PROGRAM Encoder
VAR
	//Encoder1 : Link to EL5001
	nRawData 		: REAL;
	nScaling 		: REAL;
	nOffset 		: REAL;
	nVoltage 		: REAL;
	testEncoder		: sEncoder;
	sScalingTable 	: ARRAY[0..2] OF WSTRING := ["Stacker Table WAN", "WT3 WAN"];
	iScaleTable		: INT := 0;
END_VAR



IF iScaleTable=0 THEN
	nScaling := 0.0004224;
ELSIF  iScaleTable=1 THEN
	nScaling := 0.0002636080;
ELSE
	nScaling := 0.0004224;
END_IF
 
//nCounter := UDINT_TO_REAL(Encoder1.
//testEncoder.bInputToggle := TRUE;
nVoltage := UDINT_TO_REAL(testEncoder.uCounter) * nScaling + nOffset;
	
(*
IF Module_IO.iBypassSwitch THEN
	testEncoder.bInputToggle := TRUE;
	nVoltage := UDINT_TO_REAL(testEncoder.uCounter) * nScaling;
ELSE
	testEncoder.bInputToggle := FALSE;
END_IF
*)

END_PROGRAM

(* stored: Version 1.1.0.1, ProductVersion 3.1.4024.11
   POU Encoder: Id {30275c88-29ac-483c-a832-a56134260256}, SpecialFunc None *)
